FUNCTION_BLOCK FB_MotionAxisStageNC IMPLEMENTS I_MotionAxisStage
VAR
END_VAR


METHOD FB_Init: BOOL
VAR_INPUT
    bInitRetains: BOOL; // TRUE: the retain variables are initialized (reset warm / reset cold)
    bInCopyCode: BOOL;  // TRUE: the instance will be copied to the copy code afterward (online change)

    MotionAxis : I_MotionAxis;
END_VAR
END_METHOD

END_FUNCTION_BLOCK

(* stored: Version 1.1.0.1
   POU FB_MotionAxisStageNC: Id {45435f10-a0b6-484c-acad-b1f8933a6e64}, SpecialFunc None
   Method FB_Init: Id {49583e53-ba6b-447c-9a31-a37b331ea095} *)
